ABB RobotStudio station: P1_2.rsstnx

Station P1_2 (saved by RobotStudio 24.4.11080.0)
Controller Controlador1
  mechanical unit ROB_1: IRB120_3_58__01, 6 joints, base frame (0, 0, 0) mm
Layout (positions relative to the parent item):
  - Pieza_4 [part], size 5 x 30 x 60 mm
  - Pieza_5 [part], size 5 x 30 x 60 mm
  - Pieza_3 [part], size 60 x 40 x 50 mm
  - Pinza [mechanism, from Components\Pinza.rslib] at (302, 0, 558) mm, rotated rx -180 ry 0 rz 90 deg; joint values [0, 0] (rad or m)
  - IRB120_3_58__01 [mechanism, from %ABB.RobotStudio.Models.IRB120%\IRB120_3_58_G_01.rslib] at (0, 0, 0) mm; joint values [0, 0, 0, 0, 1.5708, 1.5708] (rad or m)
  - Pieza_7 [part] at (-1036.1, 760.15, 825.85) mm, size 40 x 40 x 80 mm
Attachment: Pinza is attached to IRB120_3_58__01 / Link6
EventTableEntry 1200: ActivationMode=1, Cyclic=false, Group=, Trigger=DO_Pinza 1201, Actions=[EventTableActionMechanicalPose 1202, EventTableActionAttach 1203], Comment=
EventTableTriggerIO 1201: Operator=0, IOValue=[1], IRC5Controller=? -1, SignalSource=Controlador1 1228
EventTableActionMechanicalPose 1202: VirtualSignal=, Mechanism=Pinza 2420, ToPoseName=Pinza_cerrada, VirtualSignalValue=[1]
EventTableActionAttach 1203: MountObject=false, FlangeIndext=0, FindNearest=true, AttachmentParent=Pinza 2420, AttachmentChild=? -1, Offset=[X=1, Y=0, Z=0, W=0, X=0, Y=1, Z=0, W=0, X=0, Y=0, Z=1, W=0, X=0, Y=0, Z=0, W=1]
EventTableTriggerIO 1204: Operator=0, IOValue=[1], IRC5Controller=? -1, SignalSource=Controlador1 1228
EventTableTriggerIO 1205: Operator=0, IOValue=[1], IRC5Controller=? -1, SignalSource=Controlador1 1228
EventTableTriggerIO 1206: Operator=0, IOValue=[1], IRC5Controller=? -1, SignalSource=Controlador1 1228
EventTableTriggerIO 1207: Operator=0, IOValue=[1], IRC5Controller=? -1, SignalSource=Controlador1 1228
EventTableTriggerIO 1208: Operator=0, IOValue=[1], IRC5Controller=? -1, SignalSource=Controlador1 1228
EventTableTriggerIO 1209: Operator=0, IOValue=[1], IRC5Controller=? -1, SignalSource=Controlador1 1228
EventTableTriggerIO 1210: Operator=0, IOValue=[1], IRC5Controller=? -1, SignalSource=Controlador1 1228
EventTableTriggerIO 1211: Operator=0, IOValue=[1], IRC5Controller=? -1, SignalSource=Controlador1 1228
EventTableTriggerIO 1212: Operator=0, IOValue=[1], IRC5Controller=? -1, SignalSource=Controlador1 1228
EventTableEntry 1213: ActivationMode=1, Cyclic=false, Group=, Trigger=DO_Pinza 1214, Actions=[EventTableActionMechanicalPose 1215, EventTableActionDetach 1216], Comment=
EventTableTriggerIO 1214: Operator=0, IOValue=[0], IRC5Controller=? -1, SignalSource=Controlador1 1228
EventTableActionMechanicalPose 1215: VirtualSignal=, Mechanism=Pinza 2420, ToPoseName=Pinza_abierta, VirtualSignalValue=[1]
EventTableActionDetach 1216: AttachmentParent=Pinza 2420, AttachmentChild=? -1
EventTableTriggerIO 1217: Operator=0, IOValue=[0], IRC5Controller=? -1, SignalSource=Controlador1 1228
EventTableTriggerIO 1218: Operator=0, IOValue=[0], IRC5Controller=? -1, SignalSource=Controlador1 1228
EventTableTriggerIO 1219: Operator=0, IOValue=[0], IRC5Controller=? -1, SignalSource=Controlador1 1228
EventTableTriggerIO 1220: Operator=0, IOValue=[0], IRC5Controller=? -1, SignalSource=Controlador1 1228
EventTableTriggerIO 1221: Operator=0, IOValue=[0], IRC5Controller=? -1, SignalSource=Controlador1 1228
EventTableTriggerIO 1222: Operator=0, IOValue=[0], IRC5Controller=? -1, SignalSource=Controlador1 1228
EventTableTriggerIO 1223: Operator=0, IOValue=[0], IRC5Controller=? -1, SignalSource=Controlador1 1228
EventTableTriggerIO 1224: Operator=0, IOValue=[0], IRC5Controller=? -1, SignalSource=Controlador1 1228
EventTableTriggerIO 1225: Operator=0, IOValue=[0], IRC5Controller=? -1, SignalSource=Controlador1 1228
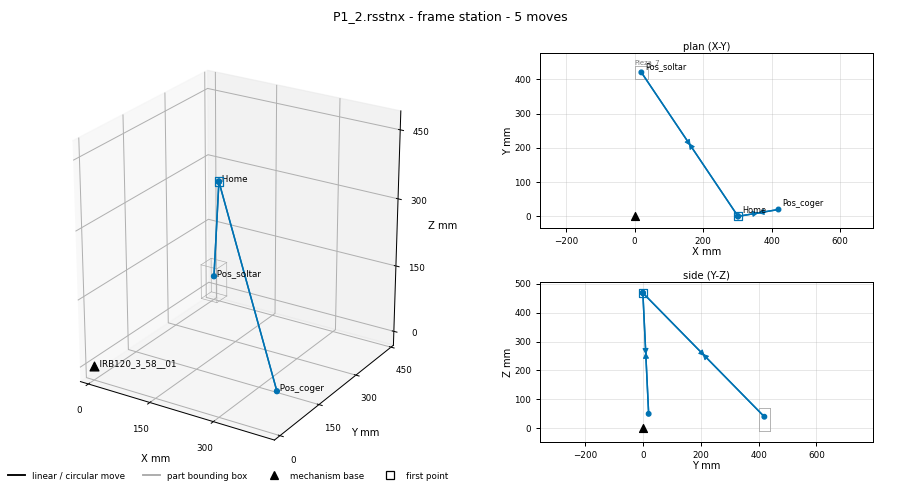
[picture p0: tool path of P1_2.rsstnx in frame station, 5 of 5 moves have a stored position in this frame; points joined in program order, loops and branches not executed]
Targets, tools, work objects and paths stored in the station, written as RAPID:
! task T_ROB1
MODULE CalibData
  PERS tooldata Pinza:=[TRUE,[[0,0,90],[1,0,0,0]],[0.5,[0,0,50],[1,0,0,0],0,0,0]];
ENDMODULE

! task T_ROB1
MODULE Module1
  CONST robtarget Home:=[[302,0,468],[0,0.707106781,0.707106781,0],[0,0,1,0],[9E+09,9E+09,9E+09,9E+09,9E+09,9E+09]];
  CONST robtarget Pos_coger:=[[420,20,50],[0,0.707106781,0.707106781,0],[0,0,1,0],[9E+09,9E+09,9E+09,9E+09,9E+09,9E+09]];
  CONST robtarget Pos_soltar:=[[20,420,40],[0,0.707106781,0.707106781,0],[0,0,1,0],[9E+09,9E+09,9E+09,9E+09,9E+09,9E+09]];
  PROC Path_10()
    MoveL Home,v200,fine,Pinza\WObj:=wobj0;
    MoveL Pos_coger,v200,fine,Pinza\WObj:=wobj0;
    SetDO DO_Pinza,1;
    WaitTime 1;
    MoveL Home,v200,fine,Pinza\WObj:=wobj0;
    MoveL Pos_soltar,v200,fine,Pinza\WObj:=wobj0;
    SetDO DO_Pinza,0;
    WaitTime 1;
    MoveL Home,v1000,z100,Pinza\WObj:=wobj0;
  ENDPROC
ENDMODULE

